TYPE ST_Machine_Service :
STRUCT
	GC_Service : ST_GC_Service;
END_STRUCT
END_TYPE

(* stored: Version 1.1.0.1, ProductVersion 3.1.4026.18
   DUT ST_Machine_Service: Id {eceae64e-ada9-4202-95e3-8ac8592a3afb} *)
